{attribute 'qualified_only'}
VAR_GLOBAL
	
//Længder af arme og afstande:
	L0Full	: REAL := 0.250;
	L0		: REAL := 0.125; //husk dette er den halve
	L1		: REAL := 0.620;
	L2		: REAL := 0.620;
	L3		: REAL := 0.745;
	L4		: REAL := 0.745;
	
	
END_VAR

(* stored: Version 1.1.0.1, ProductVersion 3.1.4024.12
   GVL GVL_LenghtData: Id {53899a9f-ee3a-4db8-8806-95bca6bca10c} *)
